FUNCTION "logger.warning_3" : Void
{ S7_Optimized_Access := 'TRUE' }
VERSION : 0.1
   VAR_INPUT
      msg : String;   // message for logging
      value_0 : String;   // additional value 0
      value_1 : String;   // additional value 1
      value_2 : String;   // additional value 2
   END_VAR

   VAR_TEMP
      str : String;
   END_VAR


BEGIN
	IF MAX_USINT(IN1 := "logger".config_in_block.level, IN2 := "logger".global_logger_level) >
	    "LoggerLevels".WARNING THEN
	    RETURN;
	END_IF;

	#str := '';
	#str := CONCAT_STRING(IN1 := #str, IN2 := #msg);
	#str := CONCAT_STRING(IN1 := #str, IN2 := '$t');
	#str := CONCAT_STRING(IN1 := #str, IN2 := #value_0);
	#str := CONCAT_STRING(IN1 := #str, IN2 := '$t');
	#str := CONCAT_STRING(IN1 := #str, IN2 := #value_1);
	#str := CONCAT_STRING(IN1 := #str, IN2 := '$t');
	#str := CONCAT_STRING(IN1 := #str, IN2 := #value_2);

	"logger._log"(level := "LoggerLevels".WARNING,
	              msg := #str
	);

END_FUNCTION

